// TIA Portal V17 export
// export: Created 2025-03-07T09:19:20.9560954Z, ExportSetting WithDefaults, DisplayName Totally Integrated Automation Portal, DisplayVersion V17 Update 8, DisplayName TIA Portal Openness, DisplayVersion V17 Update 8, DisplayName TIA Portal Version Control Interface, DisplayVersion V17, DisplayName SINAMICS Startdrive Advanced, DisplayVersion V17 SP2, DisplayName SINAMICS Startdrive G110M, G120, G120C, G120D, G120P, G115D, DisplayVersion V17 SP2, DisplayName SINAMICS Startdrive G130, G150, S120, S150, SINAMICS MV, S210, DisplayVersion V17 SP2, DisplayName STEP 7 Professional, DisplayVersion V17 Update 8, DisplayName SINUMERIK ONE STEP 7 Toolbox, DisplayVersion V17 Update 12, DisplayName SINUMERIK 840D sl STEP 7 Toolbox, DisplayVersion V17 Update 12, DisplayName STEP 7 Safety, DisplayVersion V17 Update 6, DisplayName WinCC Advanced, DisplayVersion V17 Update 8
DATA_BLOCK "DB7240_HARDWARE_SOFTWARE_ENABLE_DISABLE"   // DB7240
{ S7_Optimized_Access := 'FALSE'; DB_Accessible_From_OPC_UA := 'FALSE' }
AUTHOR : ETXETAR
VERSION : 1.0
// stored: AutoNumber false, DBAccessibleFromOPCUA false, DBAccessibleFromWebserver true, IsOnlyStoredInLoadMemory false, IsWriteProtectedInAS false
   VAR RETAIN
      DISABLE_FIXTURE : Struct
         SW_GENERAL_CONDITIONS : Bool;   // GENERAL CONDITIONS FOR GANTRY / SOFTWARE GENERAL CONDITIONS
         UNIT_01_FIX_1_4_ENABLE : Bool;   // UNIT 01 FIXTURE 1 & 4 ENABLE
         UNIT_01_FIX_2_3_ENABLE : Bool;   // UNIT 01 FIXTURE 2 & 3 ENABLE
         UNIT_02_FIX_1_4_ENABLE : Bool;   // UNIT 02 FIXTURE 1 & 4 ENABLE
         UNIT_02_FIX_2_3_ENABLE : Bool;   // UNIT 02 FIXTURE 2 & 3 ENABLE
         SW_UNIT_01_FIX_1_4_ENABLE_REQUEST : Bool;   // ENABLE REQUEST FOR GANTRY FIXTURE 1 / SOFTWARE UNIT 01 FIXTURE 1 & 4 ENABLE REQUEST
         SW_UNIT_01_FIX_1_4_DISABLE_REQUEST : Bool;   // DISABLE REQUEST FOR GANTRY FIXTURE 1 / SOFTWARE UNIT 01 FIXTURE 1 & 4 DISABLE REQUEST
         SW_UNIT_01_FIX_2_3_ENABLE_REQUEST : Bool;   // ENABLE REQUEST FOR GANTRY FIXTURE 2 / SOFTWARE UNIT 01 FIXTURE 2 & 3 ENABLE REQUEST
         SW_UNIT_01_FIX_2_3_DISABLE_REQUEST : Bool;   // DISABLE REQUEST FOR GANTRY FIXTURE 2 / SOFTWARE UNIT 01 FIXTURE 2 & 3 DISABLE REQUEST
         SW_UNIT_01_FIX_ENABLE_DISABLE_REQUEST : Bool;   // SOFTWARE UNIT 01 FIXTURE ENABLE DISABLE REQUEST
         SW_UNIT_02_FIX_1_4_ENABLE_REQUEST : Bool;   // ENABLE REQUEST FOR GANTRY FIXTURE 1 / SOFTWARE UNIT 02 FIXTURE 1 & 4 ENABLE REQUEST
         SW_UNIT_02_FIX_1_4_DISABLE_REQUEST : Bool;   // DISABLE REQUEST FOR GANTRY FIXTURE 1 / SOFTWARE UNIT 02 FIXTURE 1 & 4 DISABLE REQUEST
         SW_UNIT_02_FIX_2_3_ENABLE_REQUEST : Bool;   // ENABLE REQUEST FOR GANTRY FIXTURE 2 / SOFTWARE UNIT 02 FIXTURE 2 & 3 ENABLE REQUEST
         SW_UNIT_02_FIX_2_3_DISABLE_REQUEST : Bool;   // DISABLE REQUEST FOR GANTRY FIXTURE 2 / SOFTWARE UNIT 02 FIXTURE 2 & 3 DISABLE REQUEST
         SW_UNIT_02_FIX_ENABLE_DISABLE_REQUEST : Bool;   // SOFTWARE UNIT 02 FIXTURE ENABLE DISABLE REQUEST
         HMI_ACCEPT_BUTTON : Bool;   // HMI ACCEPT BUTTON
         SW_UNIT_01_FIX_1_4_ENABLED : Bool;   // ENABLED FOR GANTRY FIXTURE 1 / SOFTWARE UNIT 01 FIXTURE 1 & 4 ENABLED
         SW_UNIT_01_FIX_2_3_ENABLED : Bool;   // ENABLED FOR GANTRY FIXTURE 2 / SOFTWARE UNIT 01 FIXTURE 2 & 3 ENABLED
         SW_UNIT_02_FIX_1_4_ENABLED : Bool;   // ENABLED FOR GANTRY FIXTURE 1 / SOFTWARE UNIT 02 FIXTURE 1 & 4 ENABLED
         SW_UNIT_02_FIX_2_3_ENABLED : Bool;   // ENABLED FOR GANTRY FIXTURE 2 / SOFTWARE UNIT 02 FIXTURE 2 & 3 ENABLED
         UNIT_01_FIX_1_4_DISABLE_ALARM : Bool;   // FIXTURE 1 PRESENT FAULT / UNIT 01 FIXTURE 1 & 4 DISABLE ALARM
         UNIT_01_FIX_2_3_DISABLE_ALARM : Bool;   // FIXTURE 2 PRESENT FAULT / UNIT 01 FIXTURE 2 & 3 DISABLE ALARM
         UNIT_02_FIX_1_4_DISABLE_ALARM : Bool;   // FIXTURE 1 PRESENT FAULT / UNIT 02 FIXTURE 1 & 4 DISABLE ALARM
         UNIT_02_FIX_2_3_DISABLE_ALARM : Bool;   // FIXTURE 2 PRESENT FAULT / UNIT 02 FIXTURE 2 & 3 DISABLE ALARM
         DESELECT_IN_PROGRESS : Bool;   // DESELECT IN PROGRESS / DESELECTION IN PROGRESS
         SW_ALL_FIXTURES_UNIT_01_DISABLED : Bool;   // SOFTWARE ALL FIXTURES UNIT 01 DISABLED
         SW_ALL_FIXTURES_UNIT_02_DISABLED : Bool;   // SOFTWARE ALL FIXTURES UNIT 02 DISABLED
         SW_ALL_FIXTURES_DISABLED : Bool;   // SOFTWARE ALL FIXTURES DISABLED
         SW_PULSE : Array[1..20] of Bool;
      END_STRUCT;
   END_VAR
BEGIN
END_DATA_BLOCK
